FUNCTION SPLITTING_BYTE_TO_QUARTERS
  (* Standard: 61499-1; Description: Copyright (c) 2024 HR Agrartechnik GmbH This program and the accompanying materials are made available under the terms of the Eclipse Public License 2.0 which is available at https://www.eclipse.org/legal/epl-2.0/ SPDX-License-Identifier: EPL-2.0 *)
  (* Version 1.0, 2024-02-22, franz *)
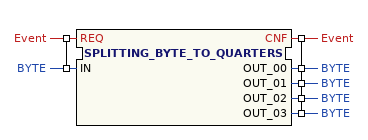
  EVENT_INPUT
    REQ WITH IN; (* Normal Execution Request *)
  END_EVENT
  EVENT_OUTPUT
    CNF WITH OUT_00, OUT_01, OUT_02, OUT_03; (* Execution Confirmation *)
  END_EVENT
  VAR_INPUT
    IN : BYTE; (* BYTE Input *)
  END_VAR
  VAR_OUTPUT
    OUT_00 : BYTE; (* QUARTER BYTE 00 *)
    OUT_01 : BYTE; (* QUARTER BYTE 01 *)
    OUT_02 : BYTE; (* QUARTER BYTE 02 *)
    OUT_03 : BYTE; (* QUARTER BYTE 03 *)
  END_VAR
  BODY IN ST:
FUNCTION SPLITTING_BYTE_TO_QUARTERS

VAR_INPUT
	IN : BYTE;    // BYTE Input
END_VAR

VAR_OUTPUT
	OUT_00 : BYTE;    // QUARTER BYTE 00
	OUT_01 : BYTE;    // QUARTER BYTE 01
	OUT_02 : BYTE;    // QUARTER BYTE 02
	OUT_03 : BYTE;    // QUARTER BYTE 03
END_VAR

(* this Function extracts the 4 QUARTER BYTE from a byte *)
OUT_00 := SHR(IN AND BYTE_QUARTER_00, SHFT_QUARTER_00);
OUT_01 := SHR(IN AND BYTE_QUARTER_01, SHFT_QUARTER_01);
OUT_02 := SHR(IN AND BYTE_QUARTER_02, SHFT_QUARTER_02);
OUT_03 := SHR(IN AND BYTE_QUARTER_03, SHFT_QUARTER_03);

END_FUNCTION
  END_BODY
END_FUNCTION
